(* IEC 61131-3 sources: logicbox/st/examples, 4 files *)

(* ---- 01-onstop.st ---- *)
PROGRAM on_stop
  VAR_EXTERNAL
    out1: BOOL;
    out2: BOOL;
  END_VAR
  out1 := TRUE;
  out2 := TRUE;
END_PROGRAM

(* ---- 01-oscillator.st ---- *)
(* multivibrator at 0.5Hz
   outputs to OUT1, OUT2 scalars
   enabled by START scalar *)
PROGRAM oscillator
  VAR_EXTERNAL
    out1: BOOL;
    out2: BOOL;
    start: BOOL;
  END_VAR

  VAR
    ton1 : TON;
    ton2 : TON;
  END_VAR

  if start then
  ton1(
       IN := not ton2.q,
       PT := T#1000ms);
  ton2(
       IN := ton1.q,
       PT := T#1000ms);
  end_if;

  out1 := ton1.q;
  out2 := not out1;
END_PROGRAM

(* ---- 03-onstop.st ---- *)
PROGRAM on_stop
  VAR_EXTERNAL
    out1: BOOL;
    out2: BOOL;
    mw1: INT;
    stop1: BOOL;
  END_VAR
  out1:=TRUE;
  out2:=TRUE;
  mw1:=0;
  stop1:=0;
END_PROGRAM

(* ---- 03-snake.st ---- *)
PROGRAM snake
  VAR_EXTERNAL
    exec: BOOL;
    inc1: INT;
    mw1: WORD;
    stop1: BOOL;
  END_VAR

  if exec then
    mw1:=SHL(mw1,1);
    if mw1=0 then
      mw1:=1;
    end_if;
  end_if;
  WHILE stop1 DO
    inc1:=inc1-1;
  END_WHILE;
  inc1:=inc1+1;
END_PROGRAM
